FUNCTION F_LrealToExcel : STRING
VAR_INPUT
	bUseComma: BOOL;
	r1:LREAL;
END_VAR
VAR
	s1:STRING;
	pos: INT;
END_VAR

//in portuguese Excel should have a comma instead of a dot
s1:=LREAL_TO_STRING(r1);
IF bUseComma THEN
	pos:= find(s1,'.');
	IF pos <> 0 THEN
		s1:=replace(s1,',',1,pos);
	END_IF	
END_IF

F_LrealToExcel:=s1;

END_FUNCTION

(* stored: Version 1.1.0.1, ProductVersion 3.1.4024.12
   POU F_LrealToExcel: Id {389078ac-b774-4274-8295-dbdfd6d59871}, SpecialFunc None *)
